PROGRAM PRG_LAS
VAR
    fb_LAS_VIS : FB_MotionStage;
    fb_LAS_D_H : FB_MotionStage;
    fb_LAS_D_V : FB_MotionStage;
    bInit : BOOl := TRUE;
	
	//EPS
	stLAS_VIS : DUT_EPS;
	fbLAS_VIS_EPS : FB_EPS;
	
	stLAS_D_H : DUT_EPS;
	fbLAS_D_H_EPS : FB_EPS;
END_VAR

IF ( bInit) THEN
    bInit := FALSE;
    Main.M36.bHardwareEnable := TRUE;
    Main.M36.bPowerSelf := TRUE;
    Main.M36.nBrakeMode := ENUM_StageBrakeMode.NO_BRAKE;
    Main.M36.nEnableMode := ENUM_StageEnableMode.DURING_MOTION;

    Main.M37.bHardwareEnable := TRUE;
    Main.M37.bPowerSelf := TRUE;
    Main.M37.nBrakeMode := ENUM_StageBrakeMode.NO_BRAKE;
    Main.M37.nEnableMode := ENUM_StageEnableMode.DURING_MOTION;

    Main.M38.bHardwareEnable := TRUE;
    Main.M38.bPowerSelf := TRUE;
    Main.M38.nBrakeMode := ENUM_StageBrakeMode.NO_BRAKE;
    Main.M38.nEnableMode := ENUM_StageEnableMode.DURING_MOTION;

END_IF
//EPS
(*
fbLAS_D_H_EPS.setDescription('Less10mm;SampleZ;PHI'); // SET DESCRITION FOR BYTE INDICATOR LABELS
//Zero is fully retracted
fbLAS_D_H_EPS.setBit(nBits:= 0, bValue:=fb_LAS_D_H.stMotionStage.fPosition<=10); 
fbLAS_D_H_EPS.setBit(nBits:= 1, bValue:=fb_LAS_D_H.stMotionStage.fPosition<=10 OR PRG_Diffractometer.fb_Diff_Z.stMotionStage.fPosition<=-20);
fbLAS_D_H_EPS.setBit(nBits:= 2, bValue:=fb_LAS_D_H.stMotionStage.fPosition<=10 OR PRG_Diffractometer.fb_Diff_Phi.stMotionStage.fPosition>0);
fbLAS_D_H_EPS(eps:=stLAS_D_H);
fb_LAS_D_H.stMotionStage.stEPSForwardEnable := stLAS_D_H; // Update Motion stage structure.

fbLAS_VIS_EPS.setDescription('IN90mm;PHIat90;Theta<10'); // SET DESCRITION FOR BYTE INDICATOR LABELS
//Zero is fully retracted
fbLAS_VIS_EPS.setBit(nBits:= 0, bValue:=fb_LAS_VIS.stMotionStage.fPosition<=5); 
fbLAS_VIS_EPS.setBit(nBits:= 1, bValue:=fb_LAS_VIS.stMotionStage.fPosition<=5 OR PRG_Diffractometer.fb_Diff_Phi.stMotionStage.fPosition<>90);
fbLAS_VIS_EPS.setBit(nBits:= 2, bValue:=fb_LAS_VIS.stMotionStage.fPosition<=5 OR PRG_Diffractometer.fb_Diff_Theta.stMotionStage.fPosition>10);
fbLAS_VIS_EPS(eps:=fbLAS_VIS_EPS);
//fb_LAS_VIS.stMotionStage.stEPSForwardEnable := fbLAS_VIS_EPS;
*)


fb_LAS_VIS(stMotionStage:=Main.M36);
fb_LAS_D_H(stMotionStage:=Main.M37);
fb_LAS_D_V(stMotionStage:=Main.M38);

END_PROGRAM

(* stored: Version 1.1.0.1, ProductVersion 3.1.4022.18
   POU PRG_LAS: Id {29e7a0d6-925c-4720-acff-704fc8fc2385}, SpecialFunc None *)
